Staubli VAL3: start.pgx

program start()
begin
  //programmation de la tache périodique
  //emissionEtat est un programme créé, et exécuté à une périodicité de 0.1s
  //taskCreateSync "emissionEtat",.1,bOverRun,emissionEtat()
  call test_ventouse()
end
